// TwinCAT 3 PLC project PLC
// ProgramVersion: 3.1.4023.0
// libraries:
//   Tc2_Standard, * (Beckhoff Automation GmbH)
//   Tc2_System, * (Beckhoff Automation GmbH)
//   Tc3_Module, * (Beckhoff Automation GmbH)
// project tree:
//   / PlcTask.TcTTO
//   POUs/ MAIN.TcPOU

CONFIGURATION PLC
    RESOURCE PLC ON TwinCAT3
        TASK PlcTask(INTERVAL := T#10ms, PRIORITY := 20);
        PROGRAM MAIN WITH PlcTask : MAIN;
    END_RESOURCE
END_CONFIGURATION

// ---- POUs/MAIN.TcPOU
PROGRAM MAIN
VAR
	FCS : BOOL := TRUE;
	FCD : BOOL := FALSE;
	FCA : BOOL := TRUE;
	FCB : BOOL := FALSE;
	START : BOOL := FALSE;
	RESET : BOOL := FALSE;
	DX : BOOL := FALSE;
	SX : BOOL := FALSE;
	SU : BOOL := FALSE;
	GIU : BOOL := FALSE;
	ALLARME : BOOL := FALSE;
	TIMER_ALLARME : TON;
	T_ALLARME : TIME := T#30s;
END_VAR

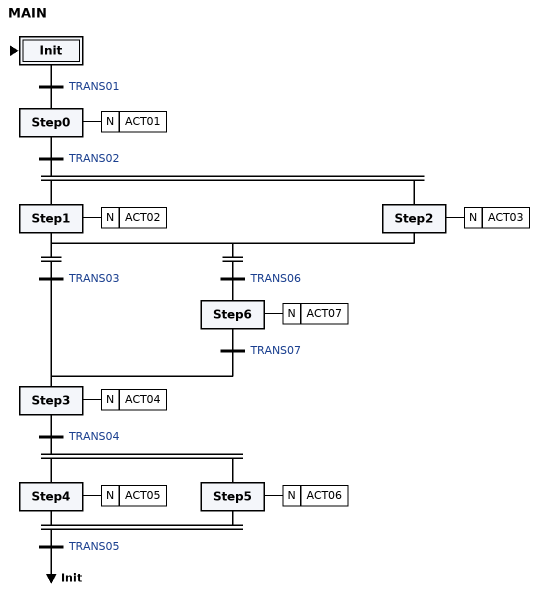
INITIAL_STEP Init:
END_STEP
TRANSITION FROM Init TO Step0
    := TRANS01;
END_TRANSITION
STEP Step0:
    ACT01(N);
END_STEP
TRANSITION FROM Step0 TO (Step1, Step2)
    := TRANS02;
END_TRANSITION
STEP Step1:
    ACT02(N);
END_STEP
STEP Step2:
    ACT03(N);
END_STEP
TRANSITION FROM (Step1, Step2) TO Step3
    := TRANS03;
END_TRANSITION
TRANSITION FROM (Step1, Step2) TO Step6
    := TRANS06;
END_TRANSITION
STEP Step6:
    ACT07(N);
END_STEP
TRANSITION FROM Step6 TO Step3
    := TRANS07;
END_TRANSITION
STEP Step3:
    ACT04(N);
END_STEP
TRANSITION FROM Step3 TO (Step4, Step5)
    := TRANS04;
END_TRANSITION
STEP Step4:
    ACT05(N);
END_STEP
STEP Step5:
    ACT06(N);
END_STEP
TRANSITION FROM (Step4, Step5) TO Init
    := TRANS05;
END_TRANSITION

ACTION ACT01:
GIU := TRUE;
END_ACTION

ACTION ACT02:
DX := TRUE;
TIMER_ALLARME(IN := TRUE, PT := T_ALLARME);
END_ACTION

ACTION ACT03:
GIU := FALSE;
SU := TRUE;
END_ACTION

ACTION ACT04:
SU := FALSE;
DX := FALSE;
GIU := TRUE;
ALLARME := FALSE;
TIMER_ALLARME(IN := FALSE , PT := T_ALLARME);
END_ACTION

ACTION ACT05:
SX := TRUE;
END_ACTION

ACTION ACT06:
SU := TRUE;
GIU := FALSE;
END_ACTION

ACTION ACT07:
ALLARME := TRUE;
TIMER_ALLARME(IN := FALSE , PT := T_ALLARME);
END_ACTION

TRANSITION TRANS01:
START AND FCA AND FCS;
END_TRANSITION

TRANSITION TRANS02:
FCB;
END_TRANSITION

TRANSITION TRANS03:
FCD AND FCA AND NOT TIMER_ALLARME.Q;
END_TRANSITION

TRANSITION TRANS04:
FCB;
END_TRANSITION

TRANSITION TRANS05:
FCA AND FCS;
END_TRANSITION

TRANSITION TRANS06:
TIMER_ALLARME.Q AND NOT FCD;
END_TRANSITION

TRANSITION TRANS07:
SU := FALSE;
DX := FALSE;
GIU := TRUE;
ALLARME := FALSE;
END_TRANSITION

END_PROGRAM
